(* Schneider Machine Expert - Basic project exercise_4.2, file version 2.9.0.0 *)
(* ProjectInformations: Name=Novo projeto *)

HARDWARE
  Cpu 0: TM221M16R/G
  EthernetConfiguration: NetworkName=M221, IpAllocationMode=FixedAddress, IpAddress=0.0.0.0, SubnetMask=0.0.0.0
  SerialLineConfiguration: Baud=Baud19200, Parity=ParityEven, DataBits=DataBits8, StopBits=StopBits1, PhysicalMedium=PhysicalMediumRs485, TransmissionMode=TransmissionModeModbusRtu, SlaveId=1, Addressing=SlaveAddressing
  MastTask: UsePeriodScanMode=false, PeriodScan=100
  FastTask: Period=255
  CpuBehavior: StartingMode=StartAsPreviousState, AutoSaveRamOnEeprom=true, WatchdogPeriod=250

SYMBOLS  (address, symbol, comment, settings)
  %M0       SIG_IN_SEN_A
  %M1       SIG_IN_SEN_B
  %M10      SIG_OUT_ATU_1_PI
  %M11      SIG_OUT_ATU_1_PM
  %M12      SIG_OUT_ATU_1_PF
  %M13      SIG_OUT_ATU_2_PI
  %M14      SIG_OUT_ATU_2_PF
  %M15      SIG_OUT_ATU_3_PI
  %M16      SIG_OUT_ATU_3_PF
  %M20      SIG_E1_E2
  %M21      SIG_E1_E3
  %M22      SIG_E2_E4
  %M23      SIG_E3_E5
  %M24      SIG_E4_E1
  %M25      SIG_E5_E1
  %X1       E1
  %X2       E2
  %X3       E3
  %X4       E4
  %X5       E5
  %TM0      FT_SIG_E2_E4  [Preset=2, Base=OneSecond]
  %TM1      FT_SIG_E4_E1  [Preset=3, Base=OneSecond]
  %TM2      FT_SIG_E1_E2E3  [Preset=1, Base=OneSecond]
  %TM3      FT_SIG_E3_E5  [Preset=2, Base=OneSecond]
  %TM4      FT_SIG_E5_E1  [Preset=3, Base=OneSecond]
  %I0.0     IN_SEN_A
  %I0.1     IN_SEN_B
  %Q0.0     OUT_ATU_1_PI
  %Q0.1     OUT_ATU_1_PM
  %Q0.2     OUT_ATU_1_PF
  %Q0.3     OUT_ATU_2_PI
  %Q0.4     OUT_ATU_2_PF
  %Q0.5     OUT_ATU_3_PI
  %Q0.6     OUT_ATU_3_PF

GRAFCET Grafcet POU
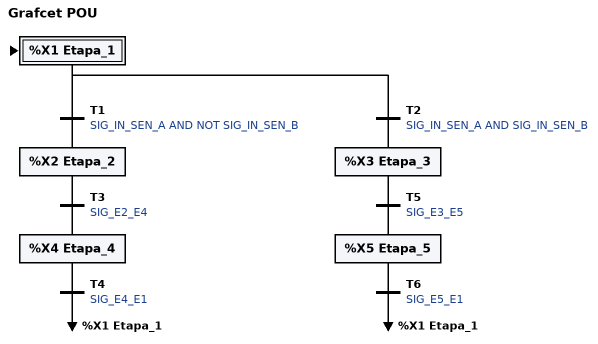
  INITIAL_STEP %X1  (* Etapa_1 *)
  STEP %X2  (* Etapa_2 *)
  STEP %X3  (* Etapa_3 *)
  STEP %X4  (* Etapa_4 *)
  STEP %X5  (* Etapa_5 *)
  TRANSITION T1 FROM %X1 TO %X2 := SIG_IN_SEN_A AND NOT SIG_IN_SEN_B;
  TRANSITION T2 FROM %X1 TO %X3 := SIG_IN_SEN_A AND SIG_IN_SEN_B;
  TRANSITION T3 FROM %X2 TO %X4 := SIG_E2_E4;
  TRANSITION T4 FROM %X4 TO %X1 := SIG_E4_E1;
  TRANSITION T5 FROM %X3 TO %X5 := SIG_E3_E5;
  TRANSITION T6 FROM %X5 TO %X1 := SIG_E5_E1;

TRANSITION T1 (%X1 -> %X2) 
  (* SectionNumber=0 *)

// Rung 0: E1_E2
  LD %M0                  (* SIG_IN_SEN_A *)
  ANDN %M1                (* SIG_IN_SEN_B *)
  ENDT
  // as ST:
  //   TRANSITION := SIG_IN_SEN_A AND NOT SIG_IN_SEN_B;

TRANSITION T2 (%X1 -> %X3) 
  (* SectionNumber=0 *)

// Rung 1: E1_E3
  LD %M0                  (* SIG_IN_SEN_A *)
  AND %M1                 (* SIG_IN_SEN_B *)
  ENDT
  // as ST:
  //   TRANSITION := SIG_IN_SEN_A AND SIG_IN_SEN_B;

TRANSITION T3 (%X2 -> %X4) 
  (* SectionNumber=0 *)

// Rung 2: E2_E4
  LD %M22                 (* SIG_E2_E4 *)
  ENDT
  // as ST:
  //   TRANSITION := SIG_E2_E4;

TRANSITION T4 (%X4 -> %X1) 
  (* SectionNumber=0 *)

// Rung 3: E4_E1
  LD %M24                 (* SIG_E4_E1 *)
  ENDT
  // as ST:
  //   TRANSITION := SIG_E4_E1;

TRANSITION T5 (%X3 -> %X5) 
  (* SectionNumber=0 *)

// Rung 4: E3_E5
  LD %M23                 (* SIG_E3_E5 *)
  ENDT
  // as ST:
  //   TRANSITION := SIG_E3_E5;

TRANSITION T6 (%X5 -> %X1) 
  (* SectionNumber=0 *)

// Rung 5: E5_E1
  LD %M25                 (* SIG_E5_E1 *)
  ENDT
  // as ST:
  //   TRANSITION := SIG_E5_E1;

POU Entradas
  (* SectionNumber=7 *)

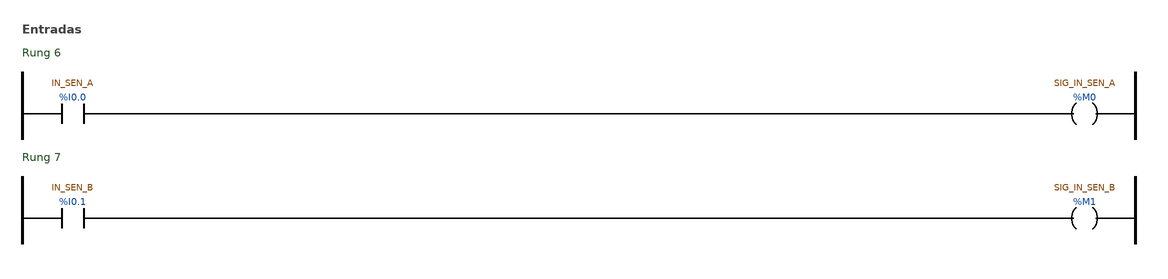

// Rung 6
  LD %I0.0                (* IN_SEN_A *)
  ST %M0                  (* SIG_IN_SEN_A *)
  // as ST:
  //   SIG_IN_SEN_A := IN_SEN_A;

// Rung 7
  LD %I0.1                (* IN_SEN_B *)
  ST %M1                  (* SIG_IN_SEN_B *)
  // as ST:
  //   SIG_IN_SEN_B := IN_SEN_B;

POU Lógicas
  (* SectionNumber=8 *)

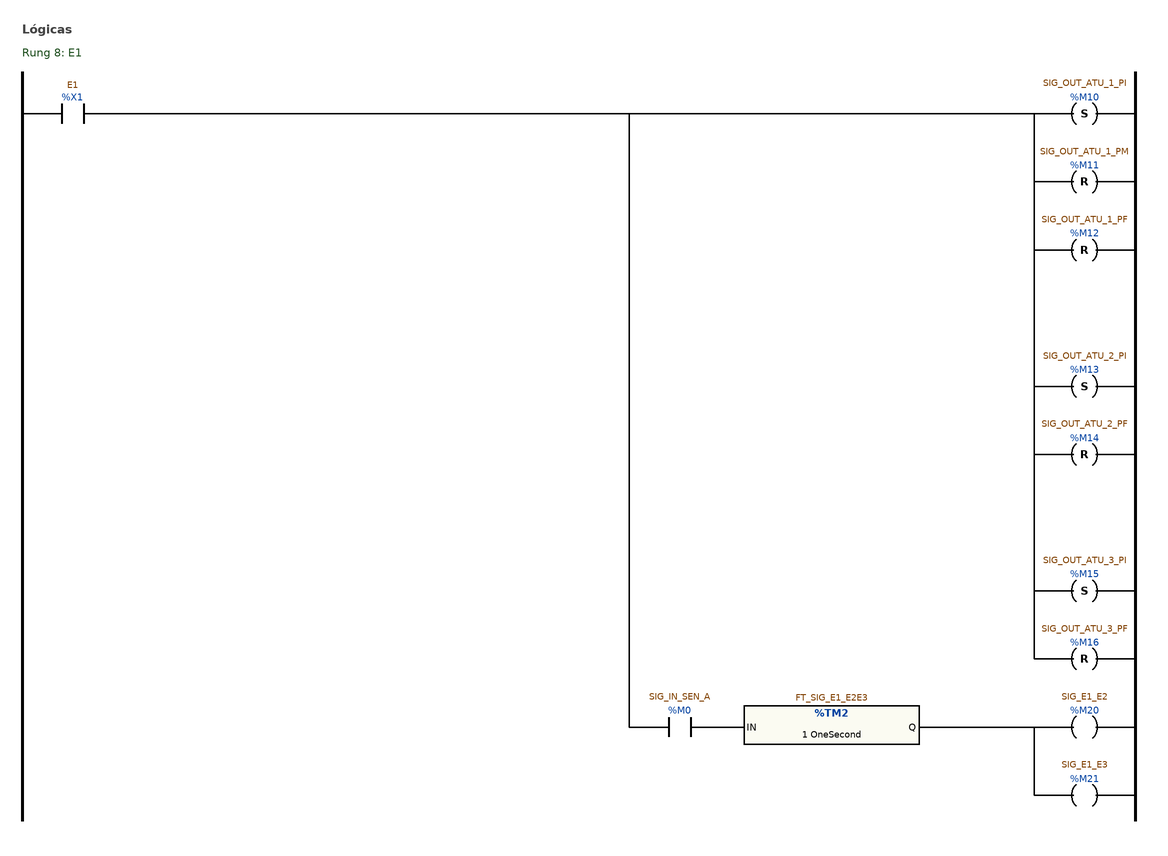

// Rung 8: E1
  LD 1
  MULTIFB
  LD 1
  AND %X1                 (* E1 *)
  ST %MW2009:X0
  LD %MW2009:X0
  S %M10                  (* SIG_OUT_ATU_1_PI *)
  R %M11                  (* SIG_OUT_ATU_1_PM *)
  R %M12                  (* SIG_OUT_ATU_1_PF *)
  S %M13                  (* SIG_OUT_ATU_2_PI *)
  R %M14                  (* SIG_OUT_ATU_2_PF *)
  S %M15                  (* SIG_OUT_ATU_3_PI *)
  R %M16                  (* SIG_OUT_ATU_3_PF *)
  BLK %TM2                (* FT_SIG_E1_E2E3 *)
  LD %MW2009:X0
  AND %M0                 (* SIG_IN_SEN_A *)
  IN
  OUT_BLK
  LD Q
  ST %M20                 (* SIG_E1_E2 *)
  ST %M21                 (* SIG_E1_E3 *)
  END_BLK
  MULTIFB
  // as ST:
  //   IF E1 THEN SIG_OUT_ATU_1_PI := TRUE; END_IF;
  //   IF E1 THEN SIG_OUT_ATU_1_PM := FALSE; END_IF;
  //   IF E1 THEN SIG_OUT_ATU_1_PF := FALSE; END_IF;
  //   IF E1 THEN SIG_OUT_ATU_2_PI := TRUE; END_IF;
  //   IF E1 THEN SIG_OUT_ATU_2_PF := FALSE; END_IF;
  //   IF E1 THEN SIG_OUT_ATU_3_PI := TRUE; END_IF;
  //   IF E1 THEN SIG_OUT_ATU_3_PF := FALSE; END_IF;
  //   FT_SIG_E1_E2E3(IN := E1 AND SIG_IN_SEN_A);
  //   SIG_E1_E2 := FT_SIG_E1_E2E3.Q;
  //   SIG_E1_E3 := FT_SIG_E1_E2E3.Q;

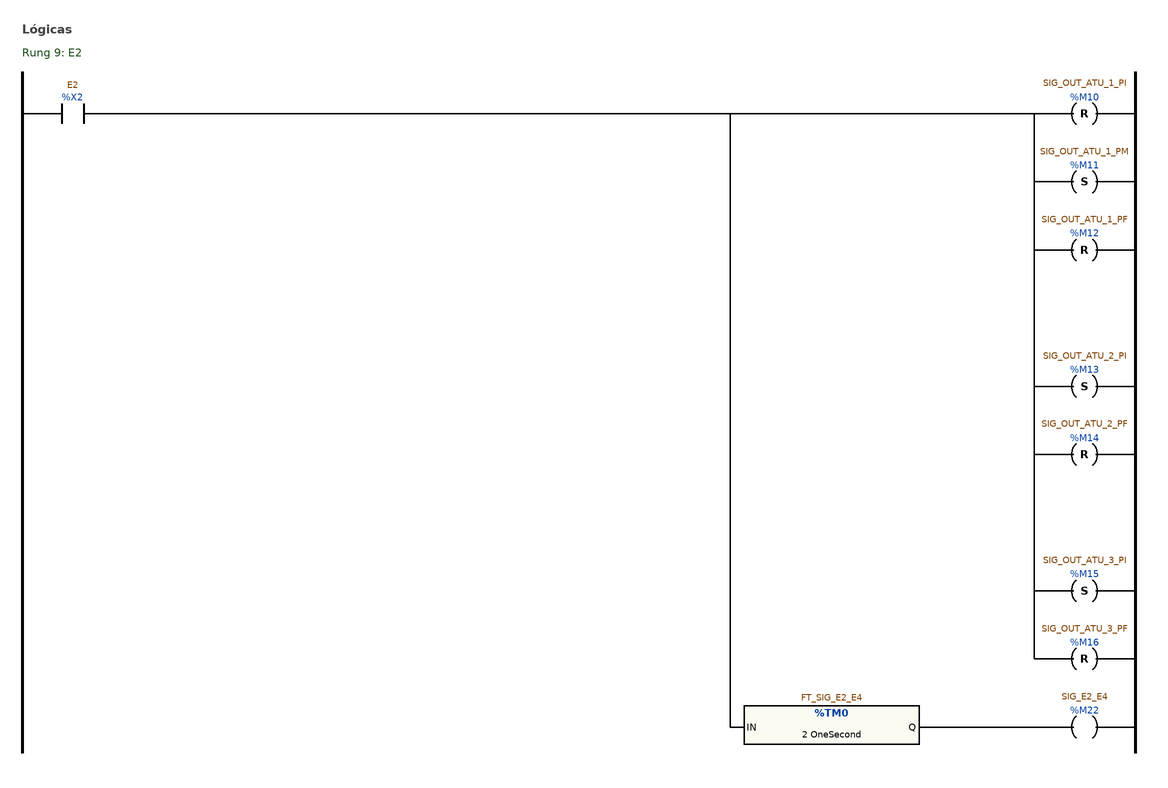

// Rung 9: E2
  LD 1
  MULTIFB
  LD 1
  AND %X2                 (* E2 *)
  ST %MW2009:X0
  LD %MW2009:X0
  R %M10                  (* SIG_OUT_ATU_1_PI *)
  S %M11                  (* SIG_OUT_ATU_1_PM *)
  R %M12                  (* SIG_OUT_ATU_1_PF *)
  S %M13                  (* SIG_OUT_ATU_2_PI *)
  R %M14                  (* SIG_OUT_ATU_2_PF *)
  S %M15                  (* SIG_OUT_ATU_3_PI *)
  R %M16                  (* SIG_OUT_ATU_3_PF *)
  BLK %TM0                (* FT_SIG_E2_E4 *)
  LD %MW2009:X0
  IN
  OUT_BLK
  LD Q
  ST %M22                 (* SIG_E2_E4 *)
  END_BLK
  MULTIFB
  // as ST:
  //   IF E2 THEN SIG_OUT_ATU_1_PI := FALSE; END_IF;
  //   IF E2 THEN SIG_OUT_ATU_1_PM := TRUE; END_IF;
  //   IF E2 THEN SIG_OUT_ATU_1_PF := FALSE; END_IF;
  //   IF E2 THEN SIG_OUT_ATU_2_PI := TRUE; END_IF;
  //   IF E2 THEN SIG_OUT_ATU_2_PF := FALSE; END_IF;
  //   IF E2 THEN SIG_OUT_ATU_3_PI := TRUE; END_IF;
  //   IF E2 THEN SIG_OUT_ATU_3_PF := FALSE; END_IF;
  //   FT_SIG_E2_E4(IN := E2);
  //   SIG_E2_E4 := FT_SIG_E2_E4.Q;

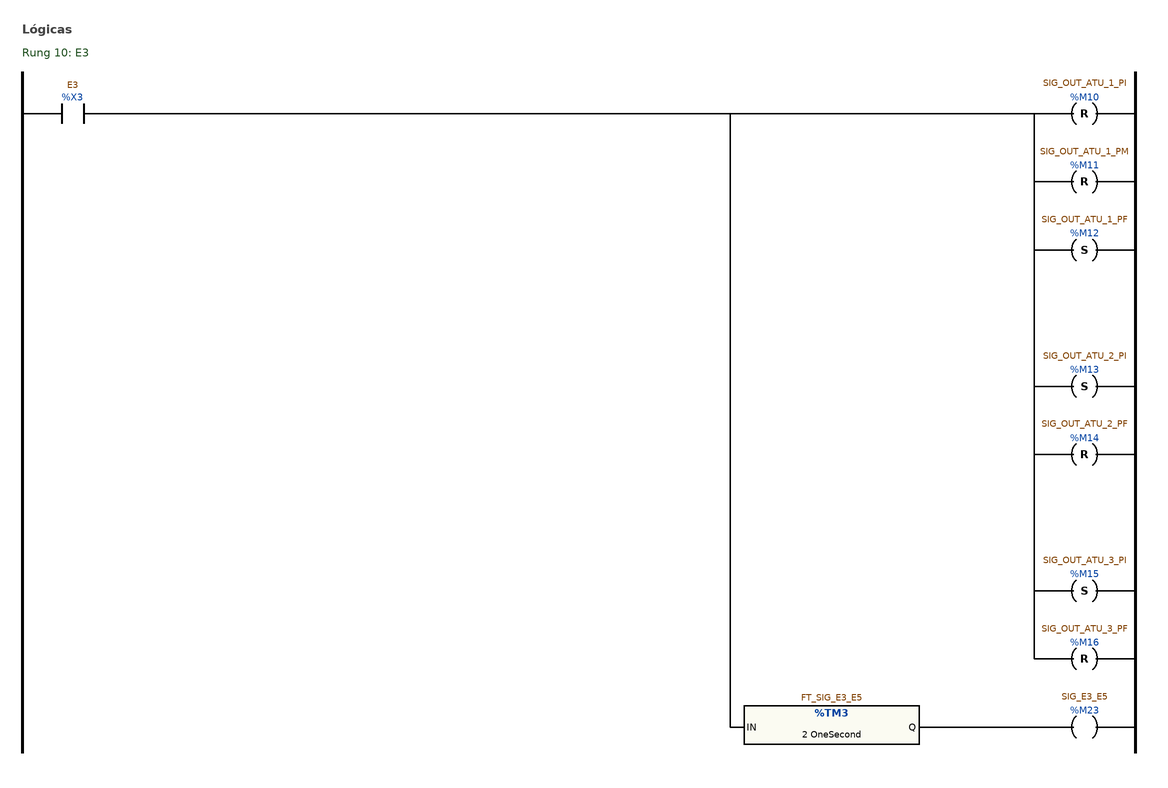

// Rung 10: E3
  LD 1
  MULTIFB
  LD 1
  AND %X3                 (* E3 *)
  ST %MW2009:X0
  LD %MW2009:X0
  R %M10                  (* SIG_OUT_ATU_1_PI *)
  R %M11                  (* SIG_OUT_ATU_1_PM *)
  S %M12                  (* SIG_OUT_ATU_1_PF *)
  S %M13                  (* SIG_OUT_ATU_2_PI *)
  R %M14                  (* SIG_OUT_ATU_2_PF *)
  S %M15                  (* SIG_OUT_ATU_3_PI *)
  R %M16                  (* SIG_OUT_ATU_3_PF *)
  BLK %TM3                (* FT_SIG_E3_E5 *)
  LD %MW2009:X0
  IN
  OUT_BLK
  LD Q
  ST %M23                 (* SIG_E3_E5 *)
  END_BLK
  MULTIFB
  // as ST:
  //   IF E3 THEN SIG_OUT_ATU_1_PI := FALSE; END_IF;
  //   IF E3 THEN SIG_OUT_ATU_1_PM := FALSE; END_IF;
  //   IF E3 THEN SIG_OUT_ATU_1_PF := TRUE; END_IF;
  //   IF E3 THEN SIG_OUT_ATU_2_PI := TRUE; END_IF;
  //   IF E3 THEN SIG_OUT_ATU_2_PF := FALSE; END_IF;
  //   IF E3 THEN SIG_OUT_ATU_3_PI := TRUE; END_IF;
  //   IF E3 THEN SIG_OUT_ATU_3_PF := FALSE; END_IF;
  //   FT_SIG_E3_E5(IN := E3);
  //   SIG_E3_E5 := FT_SIG_E3_E5.Q;

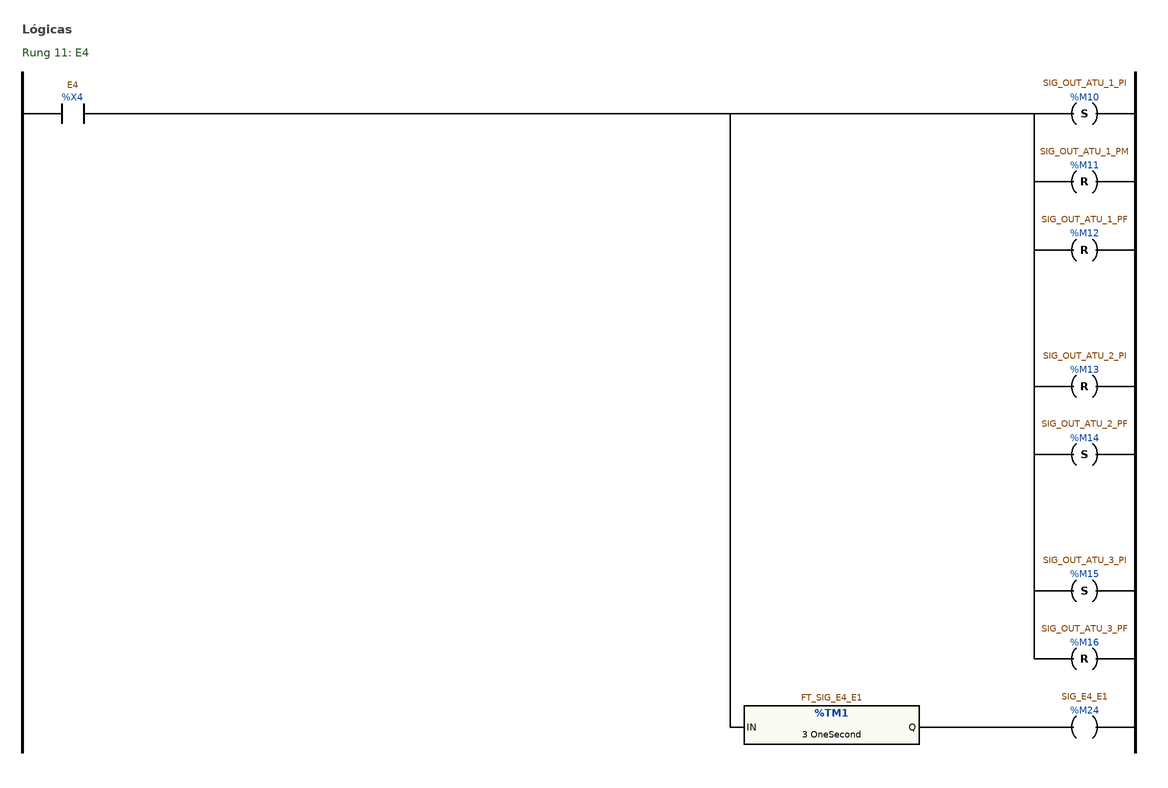

// Rung 11: E4
  LD 1
  MULTIFB
  LD 1
  AND %X4                 (* E4 *)
  ST %MW2009:X0
  LD %MW2009:X0
  S %M10                  (* SIG_OUT_ATU_1_PI *)
  R %M11                  (* SIG_OUT_ATU_1_PM *)
  R %M12                  (* SIG_OUT_ATU_1_PF *)
  R %M13                  (* SIG_OUT_ATU_2_PI *)
  S %M14                  (* SIG_OUT_ATU_2_PF *)
  S %M15                  (* SIG_OUT_ATU_3_PI *)
  R %M16                  (* SIG_OUT_ATU_3_PF *)
  BLK %TM1                (* FT_SIG_E4_E1 *)
  LD %MW2009:X0
  IN
  OUT_BLK
  LD Q
  ST %M24                 (* SIG_E4_E1 *)
  END_BLK
  MULTIFB
  // as ST:
  //   IF E4 THEN SIG_OUT_ATU_1_PI := TRUE; END_IF;
  //   IF E4 THEN SIG_OUT_ATU_1_PM := FALSE; END_IF;
  //   IF E4 THEN SIG_OUT_ATU_1_PF := FALSE; END_IF;
  //   IF E4 THEN SIG_OUT_ATU_2_PI := FALSE; END_IF;
  //   IF E4 THEN SIG_OUT_ATU_2_PF := TRUE; END_IF;
  //   IF E4 THEN SIG_OUT_ATU_3_PI := TRUE; END_IF;
  //   IF E4 THEN SIG_OUT_ATU_3_PF := FALSE; END_IF;
  //   FT_SIG_E4_E1(IN := E4);
  //   SIG_E4_E1 := FT_SIG_E4_E1.Q;

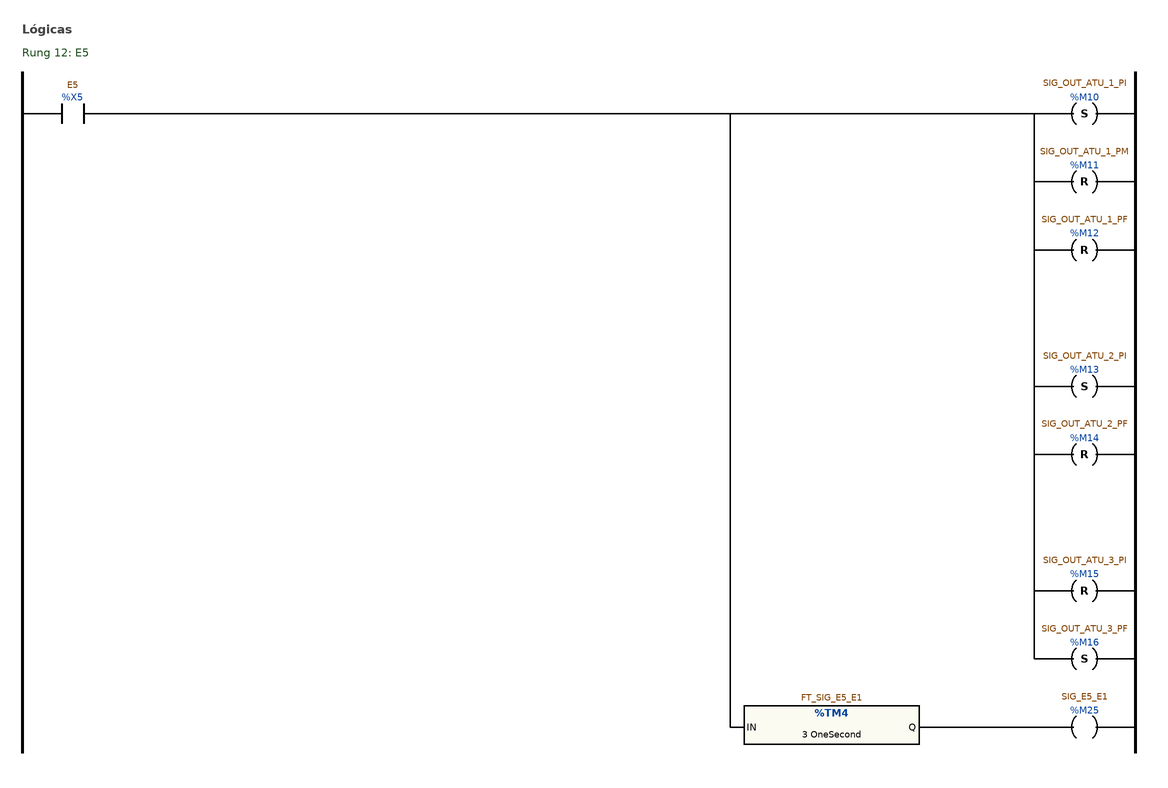

// Rung 12: E5
  LD 1
  MULTIFB
  LD 1
  AND %X5                 (* E5 *)
  ST %MW2009:X0
  LD %MW2009:X0
  S %M10                  (* SIG_OUT_ATU_1_PI *)
  R %M11                  (* SIG_OUT_ATU_1_PM *)
  R %M12                  (* SIG_OUT_ATU_1_PF *)
  S %M13                  (* SIG_OUT_ATU_2_PI *)
  R %M14                  (* SIG_OUT_ATU_2_PF *)
  R %M15                  (* SIG_OUT_ATU_3_PI *)
  S %M16                  (* SIG_OUT_ATU_3_PF *)
  BLK %TM4                (* FT_SIG_E5_E1 *)
  LD %MW2009:X0
  IN
  OUT_BLK
  LD Q
  ST %M25                 (* SIG_E5_E1 *)
  END_BLK
  MULTIFB
  // as ST:
  //   IF E5 THEN SIG_OUT_ATU_1_PI := TRUE; END_IF;
  //   IF E5 THEN SIG_OUT_ATU_1_PM := FALSE; END_IF;
  //   IF E5 THEN SIG_OUT_ATU_1_PF := FALSE; END_IF;
  //   IF E5 THEN SIG_OUT_ATU_2_PI := TRUE; END_IF;
  //   IF E5 THEN SIG_OUT_ATU_2_PF := FALSE; END_IF;
  //   IF E5 THEN SIG_OUT_ATU_3_PI := FALSE; END_IF;
  //   IF E5 THEN SIG_OUT_ATU_3_PF := TRUE; END_IF;
  //   FT_SIG_E5_E1(IN := E5);
  //   SIG_E5_E1 := FT_SIG_E5_E1.Q;

POU Saídas
  (* SectionNumber=9 *)

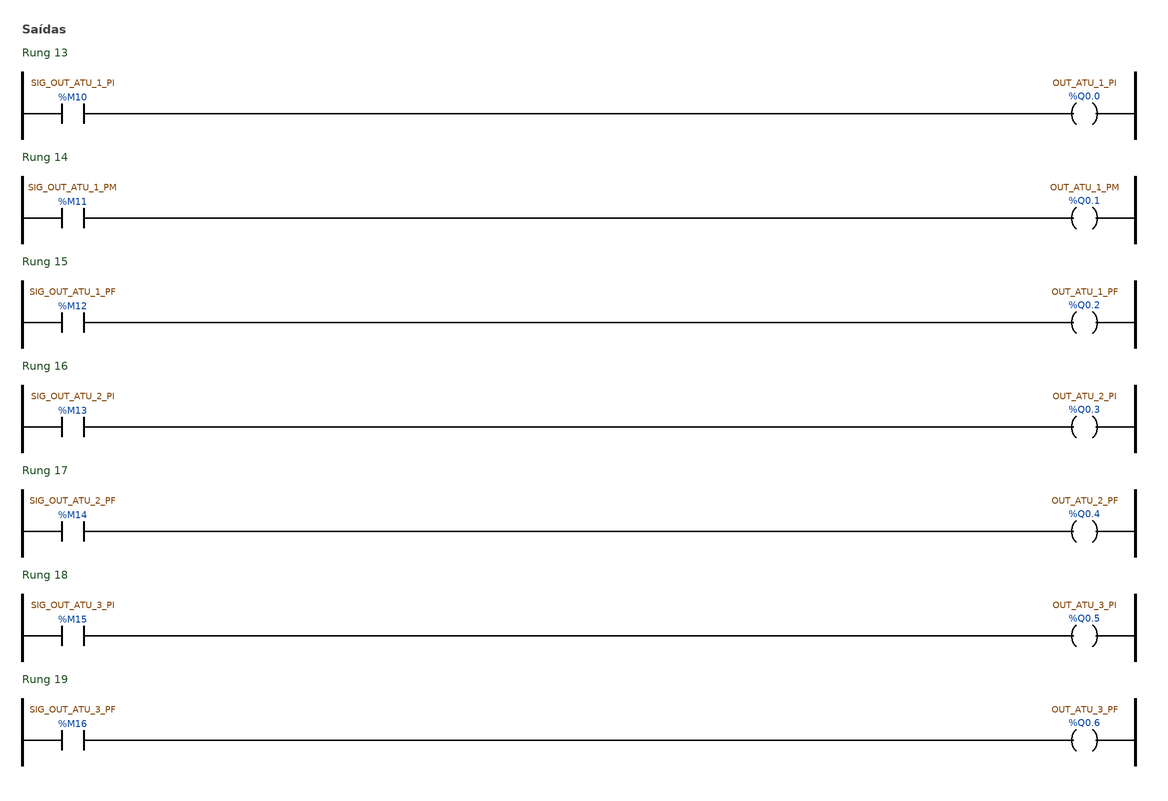

// Rung 13
  LD %M10                 (* SIG_OUT_ATU_1_PI *)
  ST %Q0.0                (* OUT_ATU_1_PI *)
  // as ST:
  //   OUT_ATU_1_PI := SIG_OUT_ATU_1_PI;

// Rung 14
  LD %M11                 (* SIG_OUT_ATU_1_PM *)
  ST %Q0.1                (* OUT_ATU_1_PM *)
  // as ST:
  //   OUT_ATU_1_PM := SIG_OUT_ATU_1_PM;

// Rung 15
  LD %M12                 (* SIG_OUT_ATU_1_PF *)
  ST %Q0.2                (* OUT_ATU_1_PF *)
  // as ST:
  //   OUT_ATU_1_PF := SIG_OUT_ATU_1_PF;

// Rung 16
  LD %M13                 (* SIG_OUT_ATU_2_PI *)
  ST %Q0.3                (* OUT_ATU_2_PI *)
  // as ST:
  //   OUT_ATU_2_PI := SIG_OUT_ATU_2_PI;

// Rung 17
  LD %M14                 (* SIG_OUT_ATU_2_PF *)
  ST %Q0.4                (* OUT_ATU_2_PF *)
  // as ST:
  //   OUT_ATU_2_PF := SIG_OUT_ATU_2_PF;

// Rung 18
  LD %M15                 (* SIG_OUT_ATU_3_PI *)
  ST %Q0.5                (* OUT_ATU_3_PI *)
  // as ST:
  //   OUT_ATU_3_PI := SIG_OUT_ATU_3_PI;

// Rung 19
  LD %M16                 (* SIG_OUT_ATU_3_PF *)
  ST %Q0.6                (* OUT_ATU_3_PF *)
  // as ST:
  //   OUT_ATU_3_PF := SIG_OUT_ATU_3_PF;
